(* Logix 5000 project; controller ECE119L_Lab6 5069-L306ERM rev 32.11; software revision 32.04 *)

TASK MainTask (continuous, watchdog 500 ms) : MainProgram

MODULES
   Local : 5069-L306ERM (5069 0, rev 32.11)
      Digital_Inputs : vendor 1 type 7 code 391 (5069 1, rev 2.1, StandardDataDriven RPI 5 ms)
      Digital_Outputs : 5069-OB16 (5069 2, rev 3.1, StandardDataDriven RPI 5 ms)
      Analog_Input : vendor 1 type 115 code 314 (5069 3, rev 2.1, StandardDataDriven RPI 100 ms)
      Analog_Inputs_2 : vendor 1 type 115 code 314 (5069 4, rev 2.1, StandardDataDriven RPI 100 ms)
      Analog_Outputs : vendor 1 type 115 code 320 (5069 5, rev 2.1, StandardDataDriven RPI 80 ms)
END_MODULES

VAR_GLOBAL   (* controller tags *)
   Screen_Out : ALIAS FOR Local:5:O.Ch00.Data;
   VDC_Input : ALIAS FOR Local:4:I.Ch00.Data;
END_VAR

PROGRAM MainProgram   (* main routine MainRoutine *)

ROUTINE MainRoutine   (* ladder *)
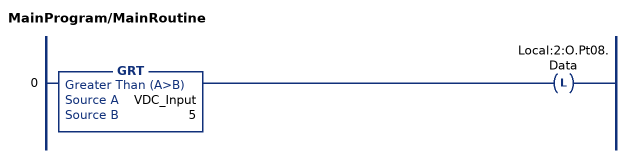
   0: GRT(VDC_Input,5)OTL(Local:2:O.Pt08.Data);
END_ROUTINE
END_PROGRAM
